Staubli VAL3: iLevel5.pgx

public program iLevel5(num& nNum[] (dimensions=1))
begin
  nNum=dioGet(iLevel5)
end
